// TIA Portal V19 export
DATA_BLOCK "DB_ExportProdData"   // DB71
{ S7_Optimized_Access := 'TRUE' }
// stored: AutoNumber false, IsOnlyStoredInLoadMemory true, MemoryReserve 100
   VAR RETAIN
      aProdData { S7_SetPoint := 'True'} : Array[0..200] of "stProductionRecord";
   END_VAR
BEGIN
   aProdData[1..2].dDate := D#2025-07-29;
   aProdData[1].todTime := TOD#13:18:42.636;
   aProdData[2].todTime := TOD#11:56:55.157;
   aProdData[1..2].sRecipeName := 'Test Carbody Shell';
   aProdData[1..2].usiProgNumber := 101;
   aProdData[1..2].sRecipeLayerTypeName := 'Putty Layer';
   aProdData[1..2].usiLayerTypeNumber := 1;
   aProdData[1].uiCbsNumber := 45;
   aProdData[2].uiCbsNumber := 46;
   aProdData[1].uiPaperUsed := 6;
   aProdData[1].tCycleTime := TOD#00:06:08.019;
   aProdData[2].tCycleTime := TOD#01:12:43.602;
END_DATA_BLOCK
